PROGRAM Utility
VAR
	LedStrip						: RgbController;
	Red								: BOOL := FALSE;
	Green							: BOOL := TRUE;
	Blue							: BOOL := FALSE;
	
	EL9227Ch1						: MDP5001_922_DEB3C1CF;
	EL9227Ch2						: MDP5001_922_DEB3C1CF;
	
	EnergyCalculator				: EnergyCalculator;
	EnergyConsumptionCostPence		: LREAL;
	
END_VAR


EnergyCalculator
(
	Voltage						:= EL9227Ch1.MDP5001_922_Input.MDP5001_922_Voltage_In / 10.0, 
	Current						:= EL9227Ch1.MDP5001_922_Input.MDP5001_922_Current / 100.0,
	PowerConsumptionAverageW	=> ,
	EnergyConsumptionTotalJ		=> , 
	EnergyConsumptionTotalkWh	=> ,
	EnergyConsumptionCostPence	=> EnergyConsumptionCostPence
);

LedStrip.SetCustom(Red, Green, Blue);

END_PROGRAM

(* stored: Version 1.1.0.1
   POU Utility: Id {44da1c63-b243-4a1f-9809-46a9666ca3d8}, SpecialFunc None *)
